FUNCTION normProjIdx: DINT
VAR_INPUT
    idx: DINT;
    size: DINT;
END_VAR
VAR
    tmp: DINT;
END_VAR

tmp := idx;
IF tmp < 0 THEN
    tmp := size + tmp;
END_IF;
normProjIdx := tmp;

END_FUNCTION

(* stored: ProductVersion 3.1.0.18, Version 1.1.0.1 *)
